{attribute 'GeneratedUsingTerminal: EL7031-0000-0016'}
{attribute addProperty BoxType "EL7031-0000-0016"}
{attribute addProperty Id "Enable_latch_extern_on_positive_edgeBOOL1Set_counterBOOL1Enable_latch_extern_on_negative_edgeBOOL1"}
{attribute addProperty CRC "4052334391"}
{attribute addProperty Size "3"}
TYPE Control_F189B737 :
STRUCT
	{attribute addProperty Name "Enable_latch_extern_on_positive_edge"}
	Enable_latch_extern_on_positive_edge : BOOL;
	{attribute addProperty Name "Set_counter"}
	Set_counter : BOOL;
	{attribute addProperty Name "Enable_latch_extern_on_negative_edge"}
	Enable_latch_extern_on_negative_edge : BOOL;
END_STRUCT
END_TYPE

(* stored: Version 1.2.0.0, ProductVersion 3.1.4024.9
   DUT Control_F189B737: Id {7c39e24d-9ff5-47a9-9619-81bb11cb688d} *)
